TYPE ST_HO_Parameter :
STRUCT

	Temp_Warmwasser         : REAL;
	Temp_Warmwasser_Max		: REAL ;
	Temp_Warmwasser_Min		: REAL;
	Temp_Heisswasser        : REAL;
	Temp_Heisswasser_Max	: REAL ;
	Temp_Heisswasser_Min	: REAL;

	AutoQuittierung			: BOOL := 0;
END_STRUCT
END_TYPE

	// Temp_Heisswasser

(* stored: Version 1.1.0.1, ProductVersion 3.1.4024.9
   DUT ST_HO_Parameter: Id {1fcb20f6-55b8-4b88-a4c9-fb12b1ac2f96} *)
